// SIMATIC S7-200 project (STEP 7-Micro/WIN), CPU 226 REL 02.00

SYMBOL_TABLE USER1
MAIN_SW          I0.0     // Main switch
LED_SW           I0.1     // LED switch
PUMP_SW          I0.2     // Pump switch
FIRST_CYCLE      SM0.1    // First cycle flag
RTC_YEAR         VB0      // RTC year
RTC_MONTH        VB1      // RTC month
RTC_DAY          VB2      // RTC day
RTC_HOUR         VB3      // RTC hour
RTC_MINUTE       VB4      // RTC month
RTC_SECOND       VB5      // RTC second
RTC_RES          VB6      // RTC reserved
RTC_WEEKDAY      VB7      // RTC weekday
SET_CLOCK        VB8      // Flag to set clock on init
CLOCK_BIT        SM0.5    // Clock seconds bit
PUMP_START_HOUR  VB20     // Pump starting hour
PUMP_END_HOUR    VB21     // Pump ending hour
SUNRISE_HOUR     VB22     // Sunrise hour
SUNDOWN_HOUR     VB23     // Sundown hour
SUNRISE_END      VB24     // Sunrise end
SUNDOWN_END      VB25     // Sundown end
TRANS_LENGTH     VW26     // Transition length
CYCLE_LENGTH     VW28     // PWM cycle length
PULSE_WIDTH      VW30     // PWM pulse length
END_SYMBOL_TABLE

ORGANIZATION_BLOCK MAIN:OB1
TITLE=AQUARIUM WATER CIRCULATION / LIGHTING CONTROLLER LOGIC
// 
// Input controls:
// I0.0 - Main switch
// I0.1 - Lighting switch
// I0.2 - Pump switch
// 
// Created by Miroslav Sergiev #25629
// Sofia University, Faculty of Mathematics and Informatics
// 2017
VAR
PWM_ERROR:BYTE;	// LB0 
END_VAR
BEGIN
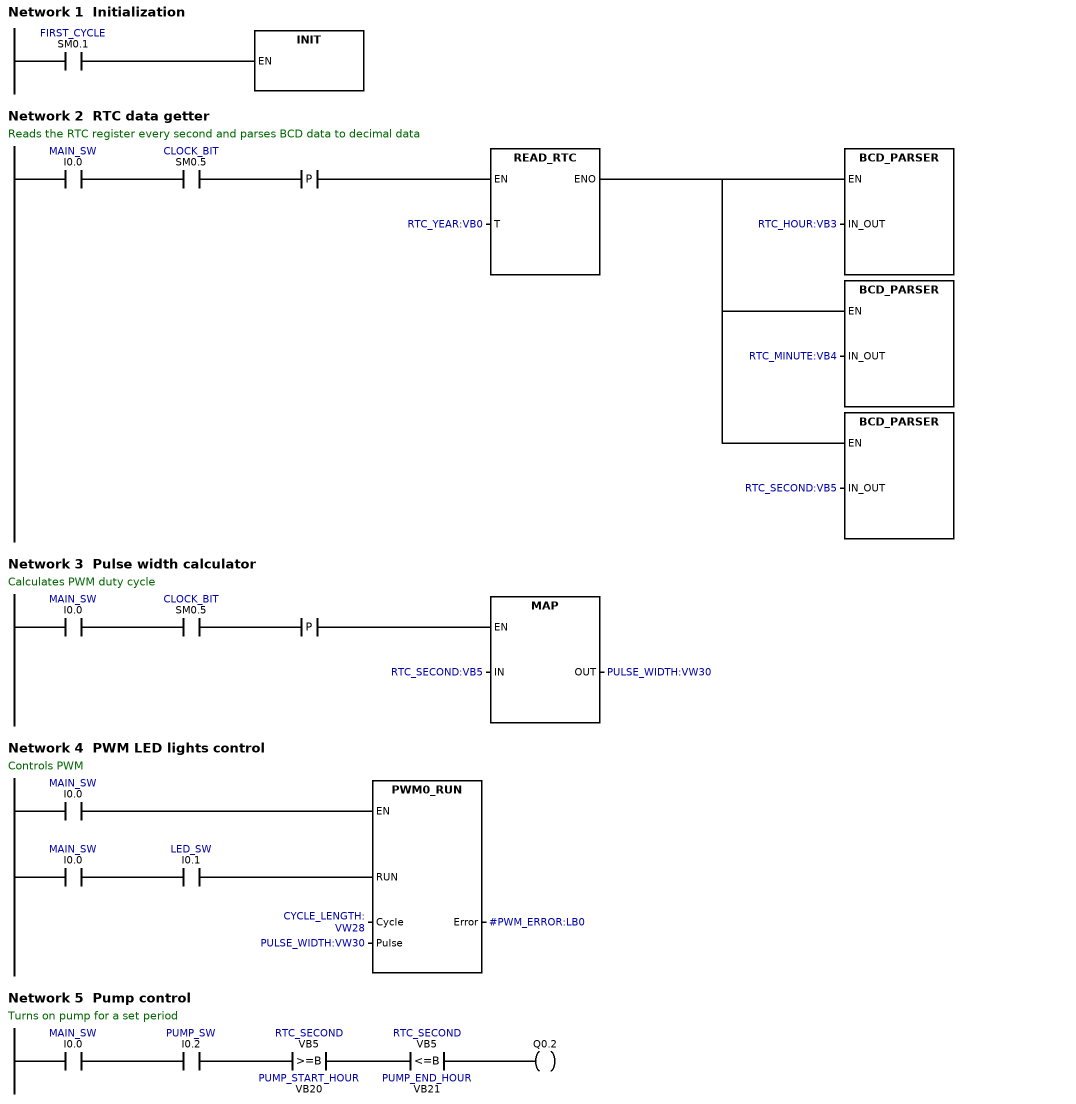
Network 1 // Initialization
LD     FIRST_CYCLE:SM0.1
CALL   INIT:SBR6
Network 2 // RTC data getter
// Reads the RTC register every second and parses BCD data to decimal data
LD     MAIN_SW:I0.0
A      CLOCK_BIT:SM0.5
EU
TODR   RTC_YEAR:VB0
AENO
CALL   BCD_PARSER:SBR2, RTC_HOUR:VB3
CALL   BCD_PARSER:SBR2, RTC_MINUTE:VB4
CALL   BCD_PARSER:SBR2, RTC_SECOND:VB5
Network 3 // Pulse width calculator
// Calculates PWM duty cycle
LD     MAIN_SW:I0.0
A      CLOCK_BIT:SM0.5
EU
CALL   MAP:SBR3, RTC_SECOND:VB5, PULSE_WIDTH:VW30
Network 4 // PWM LED lights control
// Controls PWM
LD     MAIN_SW:I0.0
=      L60.0
LD     MAIN_SW:I0.0
A      LED_SW:I0.1
=      L63.7
LD     L60.0
CALL   PWM0_RUN:SBR1, L63.7, CYCLE_LENGTH:VW28, PULSE_WIDTH:VW30, #PWM_ERROR:LB0
Network 5 // Pump control
// Turns on pump for a set period
LD     MAIN_SW:I0.0
A      PUMP_SW:I0.2
AB>=   RTC_SECOND:VB5, PUMP_START_HOUR:VB20
AB<=   RTC_SECOND:VB5, PUMP_END_HOUR:VB21
=      Q0.2
END_ORGANIZATION_BLOCK

// SBR1: protected block, not included

SUBROUTINE_BLOCK BCD_PARSER:SBR2
TITLE=BCD data parser
VAR_IN_OUT
IN_OUT:BYTE;	// LB0 Raw BCD data byte
END_VAR
VAR
LEFT_DIGIT:BYTE;	// LB1 Temporary data
RIGHT_DIGIT:BYTE;	// LB2 
LEFT_INT:INT;	// LW3 
RIGHT_INT:INT;	// LW5 
END_VAR
BEGIN
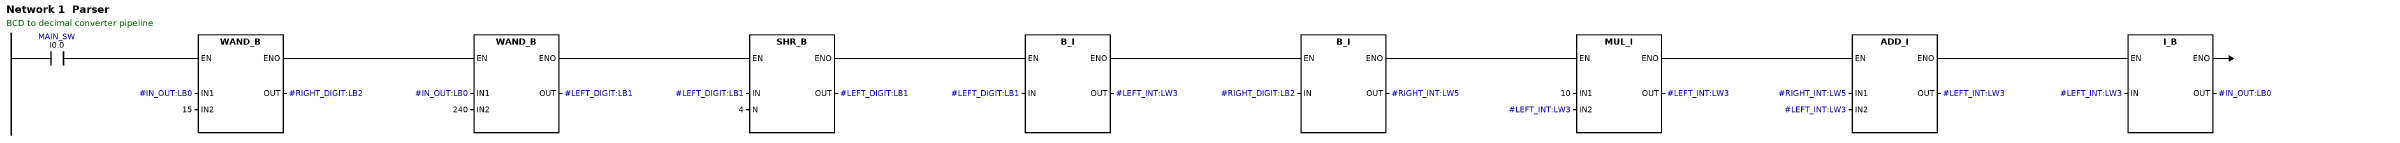
Network 1 // Parser
// BCD to decimal converter pipeline
LD     MAIN_SW:I0.0
MOVB   #IN_OUT:LB0, #RIGHT_DIGIT:LB2
AENO
ANDB   15, #RIGHT_DIGIT:LB2
AENO
MOVB   #IN_OUT:LB0, #LEFT_DIGIT:LB1
AENO
ANDB   240, #LEFT_DIGIT:LB1
AENO
SRB    #LEFT_DIGIT:LB1, 4
AENO
BTI    #LEFT_DIGIT:LB1, #LEFT_INT:LW3
AENO
BTI    #RIGHT_DIGIT:LB2, #RIGHT_INT:LW5
AENO
*I     10, #LEFT_INT:LW3
AENO
+I     #RIGHT_INT:LW5, #LEFT_INT:LW3
AENO
ITB    #LEFT_INT:LW3, #IN_OUT:LB0
END_SUBROUTINE_BLOCK

SUBROUTINE_BLOCK MAP:SBR3
TITLE=SUBROUTINE COMMENTS
VAR_INPUT
IN:BYTE;	// LB0 
END_VAR
VAR_OUTPUT
OUT:WORD;	// LW1 
END_VAR
BEGIN
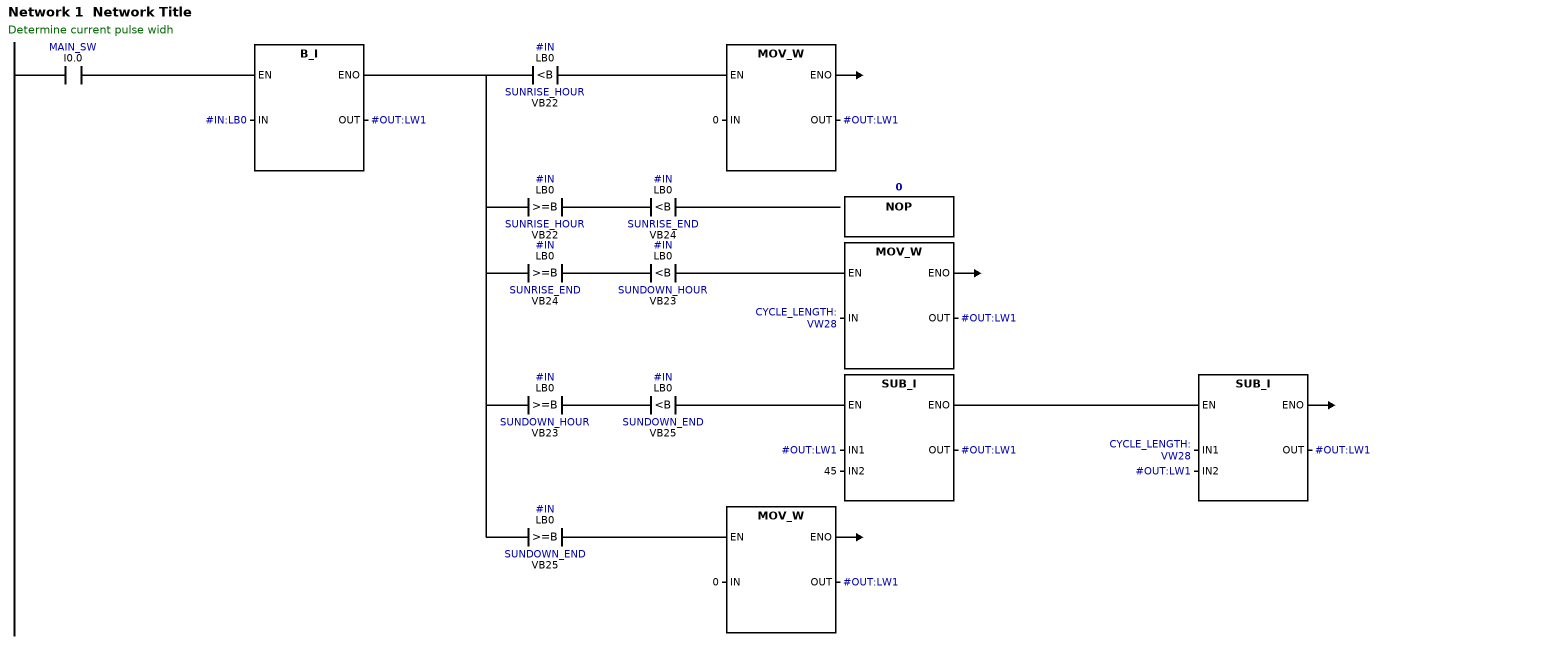
Network 1 // Network Title
// Determine current pulse widh
// (network saved uncompiled; LAD cells follow)
// row 0: c0 -| |- MAIN_SW:I0.0  c1 --  c2 [B_I EN:=power@row0, IN:=#IN:LB0, ENO=>power, OUT=>#OUT:LW1]  c3 -- v  c4 -|<B|- #IN:LB0, SUNRISE_HOUR:VB22  c5 --  c6 [MOV_W EN:=power@row0, IN:=0, ENO=>power, OUT=>#OUT:LW1]  c7 ->
// row 1: c2 [box]  c3 ^v  c6 [box]
// row 2: c3 ^v  c4 -|>=B|- #IN:LB0, SUNRISE_HOUR:VB22  c5 -|<B|- #IN:LB0, SUNRISE_END:VB24  c6 --  c7 [NOP 0 ]
// row 3: c3 ^v  c4 -|>=B|- #IN:LB0, SUNRISE_END:VB24  c5 -|<B|- #IN:LB0, SUNDOWN_HOUR:VB23  c6 --  c7 [MOV_W EN:=power@row3, IN:=CYCLE_LENGTH:VW28, ENO=>power, OUT=>#OUT:LW1]  c8 ->
// row 4: c3 ^v  c7 [box]
// row 5: c3 ^v  c4 -|>=B|- #IN:LB0, SUNDOWN_HOUR:VB23  c5 -|<B|- #IN:LB0, SUNDOWN_END:VB25  c6 --  c7 [SUB_I EN:=power@row5, IN1:=#OUT:LW1, IN2:=45, ENO=>power, OUT=>#OUT:LW1]  c8 --  c9 --  c10 [SUB_I EN:=power@row5, IN1:=CYCLE_LENGTH:VW28, IN2:=#OUT:LW1, ENO=>power, OUT=>#OUT:LW1]  c11 ->
// row 6: c3 ^v  c7 [box]  c10 [box]
// row 7: c3 ^  c4 -|>=B|- #IN:LB0, SUNDOWN_END:VB25  c5 --  c6 [MOV_W EN:=power@row7, IN:=0, ENO=>power, OUT=>#OUT:LW1]  c7 ->
// row 8: c6 [box]
END_SUBROUTINE_BLOCK

SUBROUTINE_BLOCK INIT:SBR6
TITLE=
VAR
TMP_I:WORD;	// LW0 Temporary values
END_VAR
BEGIN
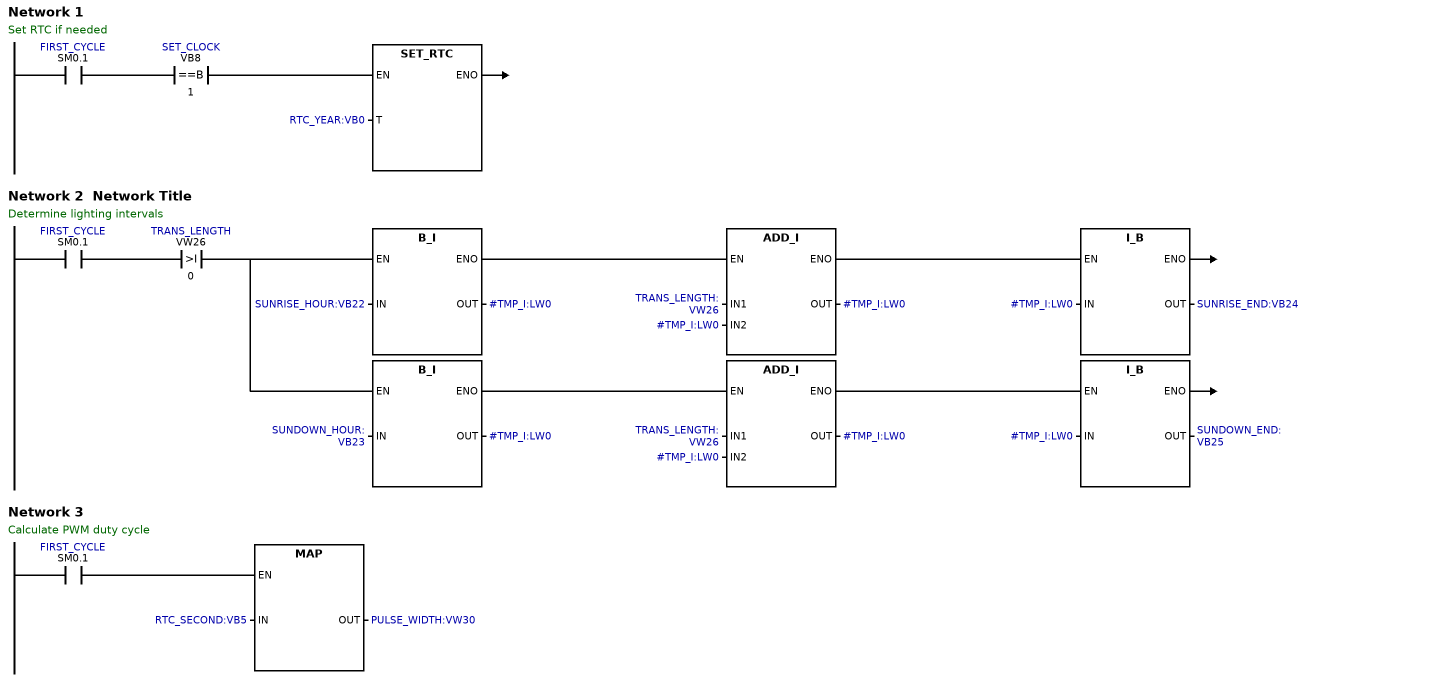
Network 1
// Set RTC if needed
LD     FIRST_CYCLE:SM0.1
AB=    SET_CLOCK:VB8, 1
TODW   RTC_YEAR:VB0
Network 2 // Network Title
// Determine lighting intervals
LD     FIRST_CYCLE:SM0.1
AW>    TRANS_LENGTH:VW26, 0
LPS
BTI    SUNRISE_HOUR:VB22, #TMP_I:LW0
AENO
+I     TRANS_LENGTH:VW26, #TMP_I:LW0
AENO
ITB    #TMP_I:LW0, SUNRISE_END:VB24
LPP
BTI    SUNDOWN_HOUR:VB23, #TMP_I:LW0
AENO
+I     TRANS_LENGTH:VW26, #TMP_I:LW0
AENO
ITB    #TMP_I:LW0, SUNDOWN_END:VB25
Network 3
// Calculate PWM duty cycle
LD     FIRST_CYCLE:SM0.1
CALL   MAP:SBR3, RTC_SECOND:VB5, PULSE_WIDTH:VW30
END_SUBROUTINE_BLOCK

DATA_BLOCK_TAB USER1
BEGIN
// PWM pulse width
         PULSE_WIDTH, 0
// PWM cycle count
         CYCLE_LENGTH, 15
// Sunrise hour
         SUNRISE_HOUR, 0
// Sundown hour
         SUNDOWN_HOUR, 45
// Transition length
         TRANS_LENGTH, 15
// Pump starting hour
         PUMP_START_HOUR, 7
// Pump ending hour
         PUMP_END_HOUR, 21
// RTC set flag
         SET_CLOCK, 1
// Current hour
         RTC_HOUR, 15
// Current minutes
         RTC_MINUTE, 23
// Current seconds
         RTC_SECOND, 48
END_DATA_BLOCK_TAB
